{attribute 'GeneratedUsingTerminal: EL2911-0000-0016'}
{attribute addProperty BoxType "EL2911-0000-0016"}
{attribute addProperty Id "FSoE_InputsFSoE_Inputs_C161D7C011FSoE_OutputsFSoE_Outputs_F73BE43A8"}
{attribute addProperty CRC "2117393216"}
{attribute addProperty Size "19"}
TYPE Module_1_FSOE_7E34DB40 :
STRUCT
	{attribute addProperty Name "FSoE_Inputs"}
	FSoE_Inputs  : FSoE_Inputs_C161D7C0;
	{attribute addProperty Name "FSoE_Outputs"}
	FSoE_Outputs  : FSoE_Outputs_F73BE43A;
END_STRUCT
END_TYPE

(* stored: Version 1.2.0.0, ProductVersion 3.1.4024.9
   DUT Module_1_FSOE_7E34DB40: Id {c0936a37-5a4b-4311-949c-b50bc6fd0656} *)
